// TIA Portal V20 export
DATA_BLOCK "HMI_Lift"   // DB9
{ S7_Optimized_Access := 'TRUE' }
// stored: MemoryReserve 100
   VAR
      Selected_Level : SInt;
      Drive_To_Sel_Lev : Bool;
      Manual_Go_Up : Bool;
      Manual_Go_Down : Bool;
      Manual_Power : Bool;
      Manual_Reset : Bool;
      Manual_Active : Bool;
   END_VAR
BEGIN
END_DATA_BLOCK
